{attribute 'qualified_only'}
{attribute 'strict'}
{attribute 'to_string'}
TYPE EPolar :
(
	Unknown := 0,
	S_Polar,
	P_Polar
);
END_TYPE

(* stored: Version 1.1.0.1, ProductVersion 3.1.4024.4
   DUT EPolar: Id {7eeb2271-5eee-442a-b359-435b7413c90e} *)
